(*
  Manages the print test/simulation. 
  - It has access to ADS_PU & ADS_Camera & JobManager 
  - It tries to do all the simulation work internally with the given references
  - Else it provides some informations & triggers for external code where this FB has no access to 
*)
FUNCTION_BLOCK FB_PrgPrint_test EXTENDS FB_BasePrint
VAR_OUTPUT
  bO_Power24V_ON  AT%Q* : BOOL;
END_VAR
VAR
  // config
  _pAdsPu : POINTER TO ST_ADS_PU;
  _pAdsSubstrate : POINTER TO ST_ADS_SUBSTRATE;
  _pAdsCamera : POINTER TO ST_ADS_CAMERA;
  
 (*test fb&data instances*)
  fb_JobManagement      : FB_JobManagement;  (*for VISU_JOB_MANAGENT*)


	(*StartUp*)
	cL_DEVS               : UINT := 1;    (*number of test PC devices*)
  
  (*helper*)
  nCtr                  : UDINT;
  sTmpPcFlags           : ST_PC_FLAGS;
  rfTStart, rfTStop     : RF_TRIG;          (*start/stop simulation trigger*)
  rfHwReady, rfTStarting: RF_TRIG;
  rfRunMachine        : RF_TRIG;
  
  _eLogLevel            : E_LogSeverity := E_LogSeverity.Info;
  _bSimPrgPrint, _bMemSimPrgPrint : BOOL;
  _bSimPrgMachine, _bMemSimPrgMachine : BOOL;
  _bSimPrgInk, _bMemSimPrgInk : BOOL;

 
  (*---- script interface ---------------*)
  bHwReady              : BOOL;             (*[status]  hardware is booted and ready (CBs in OP)*)
  bStarting             : BOOL;             (*[status]  test starting*)
  bStopping             : BOOL;             (*[status]  test stopping*)
  bRunning              : BOOL;             (*[status]  simulation runnign*)
  bStart, bStop         : BOOL;             (*[cmd]     start/stop print simulation sequence*)
  bRunMachine           : BOOL;             (*[cmd]     start machine feeder & belt*)

  (*-------------------------------------*)

END_VAR
VAR PERSISTENT
  _bEnTesting            : BOOL;
  _bEnAutoStartPrinting  : BOOL;   // automatically load a job and start printing a test pattern job
  _bEnVerboseMode        : BOOL;
  _bForceHwReady         : BOOL;
  eCameraDevice         : E_CameraDevice := E_CameraDevice.PrintMark;    (*Camera device*)
  eCameraMode           : E_CameraMode := E_CameraMode.Auto;           (*Camera mode*)
  sJobConfig            : ST_JobSettings := (*[cfg]     test job settings*)
  ( // default job
    aI_JobId := '123456780-1111-1111-1111-999999999999',
    lI_StartPage := 1,              // obsolete
    lI_EndPage := 1,                // obsolete
    lI_ImageDepth := 200_000,       // 1_127_082; //[um]
    lI_ImageWidth := 200_000,       // 455_000; //[um]
    lI_ProductionImageCount := 1,
    lI_MaintenanceImageCount := 0,
    lI_NumberOfCopies := 0,
    lI_PrintMode := 16#832200,      // bit set: 9,17,23 (13=endless)
    lI_PrePostBlankDepth := 12361,  // 292px in [um]
    lI_SubPixelResolution := 32,
    lI_ResolutionX := 600,
    aI_JobDescription := 'i1',      // endless p0
    aI_JobName := 'PRG_TEST_job'
  );
END_VAR

IF NOT bInitialized THEN RETURN; END_IF
IF NOT _bEnTesting   THEN RETURN; END_IF

//-- start / stop trigger generation
rfTStart(CLK:=bStart); rfTStop(CLK:=bStop); rfTStarting(CLK:=bStarting); rfHwReady(CLK:=bHwReady); rfRunMachine(CLK:=bRunMachine);

//-- check if hardware is ready
bHwReady := TRUE; 
FOR nCtr := 1 TO TO_UDINT(iCPr_NB_PC) DO
  IF PRG_PRINT.FB_PC[nCtr].bBoardEnable THEN
    sTmpPcFlags := PRG_PRINT.FB_PC[nCtr].sPcFlags;
    IF NOT sTmpPcFlags.bBoardInOp AND NOT _bForceHwReady THEN
      bHwReady := FALSE;
    END_IF 
  END_IF
END_FOR


// auto start stop printing 
IF    _bEnAutoStartPrinting AND rfHwReady.RT THEN bStart := TRUE;
ELSIF _bEnAutoStartPrinting AND rfHwReady.FT THEN bStop := TRUE; 
END_IF 

// starting sequence and status
bStarting := TestStartSequence();
bStopping := TestStopSequence();

// trigger actions
// - update running status
IF rfTStarting.FT THEN bRunning := TRUE;   
ELSIF rfTStop.RT  THEN bRunning := FALSE; END_IF 
// - set debug log level
IF _bEnVerboseMode THEN _eLogLevel := E_LogSeverity.Debug; 
ELSE                    _elogLevel := E_LogSeverity.Info; END_IF

(****  Job Management in ComponentsPrints ****)
fb_JobManagement(pI_Ary_Fb_Pc:= PRG_PRINT.pFB_PC^);

PROPERTY bChangedPrgSim : BOOL
GET
bChangedPrgSim := isPrgSimUpdate();
END_GET
END_PROPERTY

PROPERTY bEnterSim : BOOL
GET
bEnterSim := rfTStart.RT;
END_GET
END_PROPERTY

PROPERTY bEnTesting : BOOL
GET
bEnTesting := _bEnTesting;
END_GET
SET
_bEnTesting := bEnTesting;
END_SET
END_PROPERTY

PROPERTY bExitSim : BOOL
GET
bExitSim := rfTStop.RT;
END_GET
END_PROPERTY

PROPERTY bSimPrgInk : BOOL
GET
bSimPrgInk := _bSimPrgInk;
END_GET
SET
_bSimPrgInk := bSimPrgInk;
END_SET
END_PROPERTY

PROPERTY bSimPrgMachine : BOOL
GET
bSimPrgMachine := _bSimPrgMachine;
END_GET
SET
_bSimPrgMachine := bSimPrgMachine;
END_SET
END_PROPERTY

PROPERTY bSimPrgPrint : BOOL
GET
bSimPrgPrint := _bSimPrgPrint;
END_GET
SET
_bSimPrgPrint := bSimPrgPrint;
END_SET
END_PROPERTY

PROPERTY bStartMachine : BOOL
GET
bStartMachine := rfRunMachine.RT;
END_GET
END_PROPERTY

PROPERTY bStopMachine : BOOL
GET
bStopMachine := rfRunMachine.FT;
END_GET
END_PROPERTY

METHOD Init : BOOL
VAR_INPUT
  pAdsPu  : POINTER TO ST_ADS_PU;
  pAdsCamera : POINTER TO ST_ADS_CAMERA;
  pAdsSubstrate : POINTER TO ST_ADS_SUBSTRATE;
END_VAR
IF pAdsPu = 0 OR pAdsCamera = 0 OR pAdsSubstrate = 0 THEN
  LogError('Invalid init parameter');
  RETURN;
END_IF

_pAdsPu := pAdsPu;
_pAdsCamera := pAdsCamera;
_pAdsSubstrate := pAdsSubstrate;

(*init JobManager*)
// or default job // sJobConfig := fb_JobManagement.getJobSettings();
fb_JobManagement.Init(pI_JobSettings:=ADR(sJobConfig));

bInitialized := TRUE;
END_METHOD

METHOD isLogLevelUpdate : BOOL
VAR_OUTPUT
  eLogSeverity : E_LogSeverity;
END_VAR
VAR_INST
  oldLogSeverity : E_LogSeverity := E_LogSeverity.Info;
END_VAR
isLogLevelUpdate := SEL(oldLogSeverity <> _eLogLevel, FALSE, TRUE);
oldLogSeverity := _eLogLevel;     // remember level

eLogSeverity := _eLogLevel;
END_METHOD

METHOD PRIVATE isPrgSimUpdate : BOOL
VAR
  bChange : BOOL;
END_VAR
IF _bSimPrgInk     <> _bMemSimPrgInk     THEN _bMemSimPrgInk     := _bSimPrgInk;     bChange := TRUE; END_IF
IF _bSimPrgMachine <> _bMemSimPrgMachine THEN _bMemSimPrgMachine := _bSimPrgMachine; bChange := TRUE; END_IF
IF _bSimPrgPrint   <> _bMemSimPrgPrint   THEN _bMemSimPrgPrint   := _bSimPrgPrint;   bChange := TRUE; END_IF

isPrgSimUpdate := bChange;
END_METHOD

(*
  Load a test job
  :return: TRUE as long command is busy
*)
METHOD LoadTestJob : BOOL
VAR_INPUT
  bLoad : BOOL; 
END_VAR
VAR_INST
  bBusy : BOOL;
  tLoadTimeout : TIME;
  tExecute : TON := (PT:=T#20S);
END_VAR
IF NOT bLoad OR tExecute.Q THEN  // disable or timeout -> abort
  tExecute(IN:=FALSE);
  LoadTestJob := bBusy := FALSE;
  RETURN;
END_IF

tLoadTimeout := TO_TIME((sJobConfig.lI_ImageWidth/1000)*(sJobConfig.lI_ImageDepth/1000));             // (w[mm] * d[mm])/1000 = [s] 

tExecute(IN:=bLoad, PT:=SEL(_bForceHwReady, tLoadTimeout, T#4S));
IF NOT bBusy THEN
  // - load job
  fb_JobManagement.LoadJob(aI_AmsNetId_Io:=sC_AMSNETID_IO, pI_JobSettings:=ADR(sJobConfig));
  
  // - setup PU job
  _pAdsPu^.sI_JobSettings := sJobConfig;
  
  bBusy := TRUE;
ELSE
  bBusy := fb_JobManagement.bO_Busy; 
END_IF

LoadTestJob := bBusy;
END_METHOD

METHOD StartJob : BOOL
VAR_INPUT
END_VAR
VAR_INST
  bBusy : BOOL;
END_VAR
IF NOT _pAdsPu^.sI_Start.bI_Command THEN
  _pAdsPu^.sI_Start.bI_Command := TRUE;
  bBusy := TRUE;
ELSE    
  _pAdsPu^.sI_Start.bI_Command := FALSE;
  bBusy := FALSE;
END_IF

StartJob := bBusy;
END_METHOD

METHOD PRIVATE StopJob : BOOL
VAR_INPUT
END_VAR
VAR_INST
  bBusy : BOOL;
END_VAR
IF NOT _pAdsPu^.sI_Stop.bI_Command THEN
  _pAdsPu^.sI_Stop.bI_Command := TRUE;
  bBusy := TRUE;
ELSE    
  _pAdsPu^.sI_Stop.bI_Command := FALSE;
  bBusy := FALSE;
END_IF

StopJob := bBusy;
END_METHOD

(*
  :return: TRUE if busy
*)
METHOD PRIVATE TestStartSequence : BOOL
VAR_INPUT
END_VAR
VAR_INST
  nState			    : INT := 0;     (*start-up fsm state variable*)
  nNumDevices     : UINT;         (*loop variable*)
  nExtPcSelector  : DINT;
  tWaitJobStart   : TON := (PT:=T#4S);  (*Wait before starting job (generate pattern job)*)
END_VAR
(*-------------------------------------------*)
(* This initialize all necessary modules prior to test start*)

(*Setup Testing VarData*)
CASE nState OF

(*======> Start and Init*)
0: (*--- IDLE/START ---*)
  IF bStart THEN
    // prepare job downloader
    nNumDevices := cL_DEVS;   // set number of pc devices
    fb_JobManagement.setExtSelect(pI_Selector:=ADR(nExtPcSelector));
    nState := 1;
	END_IF

1: (*--- enter module simulations ---*)
  _bSimPrgPrint         := TRUE;
  _bSimPrgMachine       := TRUE;
  _bSimPrgInk           := TRUE;
  //_bEnVerboseMode       := TRUE;
  bO_Power24V_ON        := TRUE;
  nState := 10;
  

10: (*--- Started ---*)
  IF bStart OR nNumDevices > 0 THEN
    nState := 11;
    nExtPcSelector := nNumDevices;
  END_IF

(*======> Load initial job*)
11: (*start load default job and wait until not busy*)
  IF bHwReady OR _bForceHwReady THEN
    nState := 12;
  END_IF
  
12: (*start load default job and wait until not busy*)
  IF NOT LoadTestJob(bLoad:=TRUE) THEN 
    nNumDevices := nNumDevices - 1;
    IF nNumDevices > 0 THEN
      nState := 10;
    ELSE
      nState := 30;
    END_IF
  END_IF

(*=======> command PRG_PRINT*)
30: (*--- write job settings ---*)
  IF NOT WriteJobSettings() THEN
    nState := 40;
    tWaitJobStart(IN:=FALSE); // reset timer
    tWaitJobStart(IN:=TRUE);
  END_IF

40: (*--- wait for job generated/loaded ---*)
  IF tWaitJobStart.Q THEN
    tWaitJobStart(IN:=FALSE);
    nState := 50;
  END_IF

50: (*--- start Job ---*)
  IF NOT StartJob() THEN
    tWaitJobStart(IN:=FALSE); // reset timer
    tWaitJobStart(IN:=TRUE);
    nState := 60;
  END_IF

60: (*--- Wait for job started ---*)
  IF tWaitJobStart.Q THEN
    tWaitJobStart(IN:=FALSE);
    bRunMachine     := TRUE;            // start machine
    nState := 99;
	END_IF

98: (*Error*)
  nState := 99;

99: (*Done*)
  bStart := FALSE;
  nState := 0;

END_CASE

tWaitJobStart();
TestStartSequence := SEL(nState=0, TRUE, FALSE);
END_METHOD

(*
  :return: TRUE if busy
*)
METHOD PRIVATE TestStopSequence : BOOL
VAR_INPUT
END_VAR
VAR_INST
  nState			    : INT := 0;     (*start-up fsm state variable*)
  nNumDevices     : UINT;         (*loop variable*)
  nExtPcSelector  : DINT;
END_VAR
(*-------------------------------------------*)
(* This initialize all necessary modules prior to test start*)

(*Setup Testing VarData*)
CASE nState OF

(*======> Start and Init*)
0: (*--- IDLE/START ---*)
  IF bStop THEN
    bRunMachine := FALSE;
    //
    nNumDevices := cL_DEVS;   // set number of pc devices
    fb_JobManagement.setExtSelect(pI_Selector:=ADR(nExtPcSelector));
    nState := 1;
	END_IF

1: (*--- Started ---*)
  IF bStop OR nNumDevices > 0 THEN
    nState := 10;
    nExtPcSelector := nNumDevices;
  END_IF
  
10: (*--- for all CB ---*)
  nNumDevices := nNumDevices - 1;
  bStart := FALSE;
  IF nNumDevices > 0 THEN
    nState := 1;
  ELSE
    nState := 20;
  END_IF
  
(*======> Load initial job*)
20: (*stop job*)
  IF NOT StopJob() THEN
    nState := 60;
  END_IF
  
60: (*--- enter module simulations ---*)
  _bSimPrgPrint         := FALSE;
  _bSimPrgMachine       := FALSE;
  _bSimPrgInk           := FALSE;
  _bEnVerboseMode       := FALSE;
  bO_Power24V_ON        := FALSE;
  nState := 99;

98: (*Error*)
  nState := 99;

99: (*Done*)
  bStop := FALSE;
  nState := 0;

END_CASE

TestStopSequence := SEL(nState=0, TRUE, FALSE);
END_METHOD

(*
  :return: TRUE if busy
*)
METHOD PRIVATE WriteJobSettings : BOOL
VAR_INPUT
END_VAR

_pAdsPU^.sI_JobSettings := sJobConfig;  // set internal job settings to ads

//_pAdsSubstrate^.sI_SizeX.fI_Val := TO_REAL(sJobConfig.lI_ImageDepth);
//_pAdsSubstrate^.sI_SizeY.fI_Val := TO_REAL(sJobConfig.lI_ImageWidth);

// - setup Camera 
_pAdsCamera^.eI_CameraDevice := eCameraDevice;
_pAdsCamera^.eI_CameraMode   := eCameraMode;
//_pAdsCamera^.eI_CameraDevice := eCameraDevice; // set camera selection
//_pAdsCamera^.eI_CameraMode := eCameraMode;

// - setup substrate
_pAdsSubstrate^.aI_SubstrateName := 'A TestSubtrate equal to image dimension';
_pAdsSubstrate^.sI_SizeX.fI_Val := TO_REAL(_pAdsPu^.sI_JobSettings.lI_ImageDepth) / 1_000;  // [um] -> [mm]
_pAdsSubstrate^.sI_SizeY.fI_Val := TO_REAL(_pAdsPu^.sI_JobSettings.lI_ImageWidth) / 1_000;  // [um] -> [mm]
_pAdsSubstrate^.sI_SizeZ.fI_Val := 0;

WriteJobSettings := FALSE;
END_METHOD

END_FUNCTION_BLOCK

(* stored: Version 1.1.0.1, ProductVersion 3.1.4024.11
   POU FB_PrgPrint_test: Id {6437269a-fd39-489f-80d8-8f72b2e62aa4}, SpecialFunc None
   Folder Steps: Id {1c2bf506-7462-4584-93c3-ab8ef7ee4406}
   Property bChangedPrgSim: Id {d9c87d3f-e314-413f-a4c7-1fbddf01f857}
   Get Get: Id {af5011a4-d5a4-43b5-bedb-3d0bfb375f35}
   Property bEnterSim: Id {c5f06ca0-9a27-41e0-b448-7a64b208bc27}
   Get Get: Id {0bd501f5-8b08-4bb3-9efb-41364e272b34}
   Property bEnTesting: Id {6952b662-26c9-4f36-9192-bc40804616b2}
   Get Get: Id {53df3f35-9d66-4a48-9ac1-bafccacbd907}
   Set Set: Id {b4afae7e-b063-4e9a-882c-d2838aef5ee7}
   Property bExitSim: Id {6ef1e3c8-7b17-415d-9a6d-14f14372985b}
   Get Get: Id {3a6e1fc4-7980-4a81-aadc-858664885975}
   Property bSimPrgInk: Id {c0fa9b44-cbec-4360-9076-debc6c4c5de0}
   Get Get: Id {4d24ae91-4cb8-472c-b7ef-c4d56cef7f08}
   Set Set: Id {967e7924-ae8e-44e2-90c6-879673cec8ba}
   Property bSimPrgMachine: Id {b670674d-c113-431a-a52c-ea9542db6a53}
   Get Get: Id {d59af98d-3c71-466f-84cb-c0199474f078}
   Set Set: Id {dd8ed5e1-656f-4ca2-98c6-c2dbc5f62cdc}
   Property bSimPrgPrint: Id {d50ec45b-811f-405e-ac80-e35016b709f0}
   Get Get: Id {a37840d6-31e6-4f08-a3c8-e06f2acf46a7}
   Set Set: Id {f25ff71b-4f7f-411b-9045-cf79444fd246}
   Property bStartMachine: Id {f4faaa40-3590-4e27-9726-5ba8a58e43b5}
   Get Get: Id {2b724288-e845-4311-92e9-c4d21f268848}
   Property bStopMachine: Id {5ca955ab-5c87-4fe4-a56e-73c79214742b}
   Get Get: Id {5f359978-4746-42fb-b753-5afcdddded6b}
   Method Init: Id {64d5efce-105b-462b-a674-4598370099ea}
   Method isLogLevelUpdate: Id {c8e2138a-7774-42af-81ae-32b925ace46c}
   Method isPrgSimUpdate: Id {df7fc7cd-b95d-4d26-829f-6e040dbc207f}
   Method LoadTestJob: Id {f3876b6b-a231-42f4-b8c5-e823bd09495a}
   Method StartJob: Id {08419ff5-fef9-4c7f-a588-23b26c1ac0ff}
   Method StopJob: Id {f157481a-d9a6-4056-a7eb-17b292bab17b}
   Method TestStartSequence: Id {518534ec-20c2-4503-ab64-6616afe88650}
   Method TestStopSequence: Id {2a83d62c-0194-4737-b20b-885a814d9b26}
   Method WriteJobSettings: Id {c802bd2a-5c7d-4b77-9804-aa80ed9b6dfa} *)
